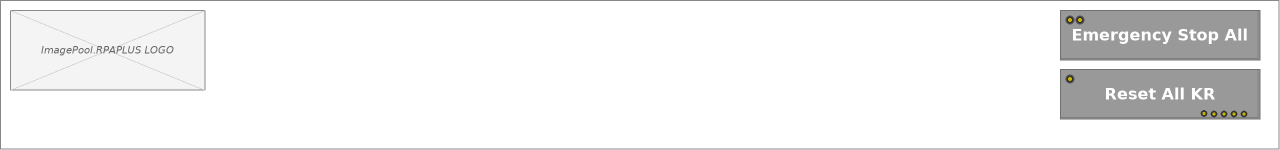
VISUALIZATION Header  // 1280x150
    Button (1060,10 200x50), "Emergency Stop All", pressed state: MAIN.btnSoftEstop
        toggle MAIN.btnSoftEstop
        OnMouseClick: execute {
            LOGFILE( sLogEvent	 := MSG.EVENT_BTN,
            		 sLogComp	 := MSG.COMP_HMI,
            		 sLogAction	 := MSG.ACTION_ESTOP,
            	 	 logFlag	 := TRUE);
        }
    Image (10,10 195x80), image: ImagePool.RPAPLUS LOGO
    Button (1060,69 200x50), "Reset All KR", pressed state: MAIN.btn_Reset or MAIN.Reset_State
        tap MAIN.btn_Reset
        OnMouseClick: execute {
            LOGFILE( sLogEvent	 := MSG.EVENT_BTN,
            		 sLogComp	 := MSG.COMP_HMI,
            		 sLogAction	 := MSG.ACTION_RESET_KUKA,
            	 	 logFlag	 := TRUE);
        }
    Lamp1 (1065,74 10x10), variable: MAIN.Reset_State, style: Lamp-Lamp1-Yellow
    Lamp1 (1200,109 8x9), variable: KR5.KR_ProgReady, style: Lamp-Lamp1-Yellow
    Lamp1 (1240,109 8x10), variable: KR1.KR_ProgReady, style: Lamp-Lamp1-Yellow
    Lamp1 (1230,109 8x10), variable: KR4.KR_ProgReady, style: Lamp-Lamp1-Yellow
    Lamp1 (1220,109 8x10), variable: KR2.KR_ProgReady, style: Lamp-Lamp1-Yellow
    Lamp1 (1210,109 8x10), variable: KR3.KR_ProgReady, style: Lamp-Lamp1-Yellow
    Lamp1 (1065,15 10x10), variable: not MAIN.btnEstop, style: Lamp-Lamp1-Yellow
    Lamp1 (1075,15 10x10), variable: MAIN.btnSoftEstop, style: Lamp-Lamp1-Yellow
END_VISUALIZATION

(* stored: Version 1.1.0.1, ProductVersion 3.1.4024.12
   Visu Header: Id {d901a921-5cec-4533-85b5-1ac952f2a093} *)
